TYPE E_TipCleaningMode :
(
	Undefined,
    Wire,
    Brush,
    WireAndBrush	
)USINT;
END_TYPE

(* stored: Version 1.1.0.1, ProductVersion 3.1.4024.5
   DUT E_TipCleaningMode: Id {bdc08032-3f7b-4df3-9cf7-f2479447c694} *)
